(* CODESYS project CtaSysSensorReCalculation_1.0.0.0.library
   Description: Sensor neu Berrechnung Library der CTA
   Version: 1.0.0.0
   Title: CtaSysSensorReCalculation
   Author: SIS
   Company: CTA
   Placeholder: CtaSysSensorReCalculation
   DocFormat: reStructuredText
   DefaultNamespace: CtaSysSensorReCalculation
   CompiledLibraryCompatibilityVersion: CODESYS V3.5 SP16 Patch 3
   LanguageModelAttribute: qualified-access-only

Project tree, tasks and I/O mapping:
  libraries: Visu Utils, 4.5.0.0 (System); Standard, 3.5.18.0 (System); CtaVisSymbols, 1.0.0.0 (CTA); VisuSymbols, 4.5.0.0 (System); CtaSysConfig, 1.0.0.2 (CTA)
  40 Visualizations/
    visualisation ValueRC
    visualisation ValueRC_QUERY
    visualisation ValueRC_BASE
  00000000-0000-0000-0000-000000000000|D:\CoDeSys\LibrariesV3\trunk\Intern\CAA\CAA Template\3.4.0.0 draft\Placeholder.xml
  00000000-0000-0000-0000-000000000000|D:\CoDeSys\LibrariesV3\trunk\Intern\CAA\CAA Template\3.2.0.3 draft\Prefix.pdf
  00000000-0000-0000-0000-000000000000|D:\CoDeSys\LibrariesV3\trunk\Intern\CAA\CAA Template\3.5.2.0 draft\Placeholder.xml
  20 Structs/
  50 Images/
  10 Documenation/
    global variables VersionHistory
    global variables readMe
  21 Interface/
    interface ITF_SENSOR_RE_CALCULATE: CALCULATET_VALUE, VALUE, UNIT
  11 Library Parameter/
  12 Konstanten/
  60 Textlisten/
  13 Globale Variablen/
  text list GlobalTextList
  5ce3da45-db07-42e7-a21c-a00fff4ed8f6|C:\Users\sis\Downloads\dip-switch.svg
  5ce3da45-db07-42e7-a21c-a00fff4ed8f6|C:\Users\sis\Downloads\lightning-bolt-circle.svg
  30 Program Organization Units/
    function block FB_SENSOR_RE_CALCULATE [ST]: CALCULATET_VALUE, VALUE, UNIT, FB_INIT
  5ce3da45-db07-42e7-a21c-a00fff4ed8f6|C:\Users\sis\Downloads\sine-wave.svg
  5ce3da45-db07-42e7-a21c-a00fff4ed8f6|C:\Users\sis\Downloads\eye.svg
  5ce3da45-db07-42e7-a21c-a00fff4ed8f6|C:\Users\sis\Downloads\lan.svg
*)

// 10 Documenation/VersionHistory
(* 

.. image:: ../../Images/CTA_Logo.jpg
   :align: right
   :width: 15% 

**Vorlage**   


============ =========== =========== ============================================
**Date**     **Version** **Author**  **Change**
------------ ----------- ----------- --------------------------------------------
04.03.2021   0.0.0.0     SIS         Vorlage erstellt

============ =========== =========== ============================================


*)
VAR_GLOBAL
    stInfo : STRING:= '0.0.0.0, Vorlage, CTA';
END_VAR

// 10 Documenation/readMe
(*

**ReadMe**
 
|	**Empfehlung**
|
|	Dokumentrieren Sie die Library für eine nachhaltige Entwicklung
|     
| *Beispiel*
| 
| Dies ist die Vorlage Library der CTA. Erstellen Sie ihre Library anhand dieser Vorlage.
*)

VAR_GLOBAL
    xReadMeDone              :   BOOL;
END_VAR

// 21 Interface/ITF_SENSOR_RE_CALCULATE
INTERFACE ITF_SENSOR_RE_CALCULATE EXTENDS __SYSTEM.IQueryInterface

PROPERTY CALCULATET_VALUE : Real
GET
END_GET
END_PROPERTY

PROPERTY VALUE : Real
SET
END_SET
END_PROPERTY

PROPERTY UNIT : STRING(5)
SET
END_SET
GET
END_GET
END_PROPERTY

END_INTERFACE

// 30 Program Organization Units/FB_SENSOR_RE_CALCULATE
FUNCTION_BLOCK FB_SENSOR_RE_CALCULATE IMPLEMENTS ITF_SENSOR_RE_CALCULATE
VAR_INPUT
	stUNIT			:	STRING(5);
END_VAR
VAR
	rValue			:	REAL;
	rCalculatet		:	REAL;
END_VAR

PROPERTY CALCULATET_VALUE : REAL
GET
rCalculatet := rValue;
CALCULATET_VALUE := rCalculatet;
END_GET
END_PROPERTY

PROPERTY VALUE : REAL
SET
rValue := VALUE;
END_SET
END_PROPERTY

PROPERTY UNIT : STRING(5)
GET
UNIT := stUNIT;
END_GET
SET
stUNIT := UNIT;
END_SET
END_PROPERTY

//FB_Init ist immer implizit verfügbar und wird primär für die Initialisierung verwendet.
//Der Rückgabewert wird nicht ausgewertet. Für gezielte Einflussnahme können Sie
//die Methoden explizit deklarieren und darin mit dem Standard-Initialisierungscode 
//zusätzlichen Code bereitstellen. Sie können den Rückgabewert auswerten.
METHOD FB_Init: BOOL
VAR_INPUT    
bInitRetains: BOOL; // TRUE: Die Retain-Variablen werden initialisiert (Reset warm / Reset kalt)    
bInCopyCode: BOOL;  // TRUE: Die Instanz wird danach in den Kopiercode kopiert (Online-Change)
_stUNIT	   : STRING(5);
END_VAR
stUNIT := _stUNIT;
END_METHOD

END_FUNCTION_BLOCK

// 40 Visualizations/ValueRC
VISUALIZATION ValueRC  // 68x12
VAR_INPUT
    ITF_SENSOR_RE_CALCULATE   :   ITF_SENSOR_RE_CALCULATE;	
END_VAR
VAR_INPUT CONSTANT
    uiTextAusrichtung   : UINT := 4;    // 0 = Oben links | 1 = Horizontal zentriert | 2 = Rechts | 4 = Vertikal zentriert | 8 = Unten
END_VAR
    Frame (0,0 68x12), invisible if: NOT __QUERYINTERFACE(ITF_SENSOR_RE_CALCULATE,ITF_SENSOR_RE_CALCULATE)
        shows ValueRC_QUERY(ITF_SENSOR_RE_CALCULATE := ITF_SENSOR_RE_CALCULATE, uiTextAusrichtung := uiTextAusrichtung)
END_VISUALIZATION

// 40 Visualizations/ValueRC_QUERY
VISUALIZATION ValueRC_QUERY  // 68x12
VAR_INPUT
    ITF_SENSOR_RE_CALCULATE   :   ITF_SENSOR_RE_CALCULATE;	
END_VAR
VAR_INPUT CONSTANT
    uiTextAusrichtung   : UINT := 4;    // 0 = Oben links | 1 = Horizontal zentriert | 2 = Rechts | 4 = Vertikal zentriert | 8 = Unten
END_VAR
    Frame (0,0 68x12)
        shows ValueRC_BASE(ITF_SENSOR_RE_CALCULATE := ITF_SENSOR_RE_CALCULATE, uiTextAusrichtung := uiTextAusrichtung)
END_VISUALIZATION

// 40 Visualizations/ValueRC_BASE
VISUALIZATION ValueRC_BASE  // 68x12
VAR_INPUT
    ITF_SENSOR_RE_CALCULATE   :   ITF_SENSOR_RE_CALCULATE;	
END_VAR
VAR_INPUT CONSTANT
    uiTextAusrichtung   : UINT := 4;    // 0 = Oben links | 1 = Horizontal zentriert | 2 = Rechts | 4 = Vertikal zentriert | 8 = Unten
END_VAR
    Textfield (0,0 68x12), "%s", text variable: CONCAT(ctaSysConfig.fcRealToString(ITF_SENSOR_RE_CALCULATE.CALCULATET_VALUE,1),TO_STRING(ITF_SENSOR_RE_CALCULATE.UNIT))
        p3718999670: uiTextAusrichtung
END_VISUALIZATION
